PROGRAM BA02PL_LineBackground
VAR
END_VAR

MAIN.stLine_BA02PL.fbLine(stLine:=MAIN.stLine_BA02PL,bMainLine:=TRUE);
MAIN.stLine_BA02PL.stStation_BA02PL01.fbStation(
				stLine:=MAIN.stLine_BA02PL,
				stStation:=MAIN.stLine_BA02PL.stStation_BA02PL01);
MAIN.stLine_BA02PL.stStation_BA02PL02.fbStation(
				stLine:=MAIN.stLine_BA02PL,
				stStation:=MAIN.stLine_BA02PL.stStation_BA02PL02);
MAIN.stLine_BA02PL.stStation_BA02PL03.fbStation(
				stLine:=MAIN.stLine_BA02PL,
				stStation:=MAIN.stLine_BA02PL.stStation_BA02PL03);
MAIN.stLine_BA02PL.stStation_BA02PL04.fbStation(
				stLine:=MAIN.stLine_BA02PL,
				stStation:=MAIN.stLine_BA02PL.stStation_BA02PL04);
MAIN.stLine_BA02PL.stStation_BA02PL05.fbStation( 
				stLine:=MAIN.stLine_BA02PL,
				stStation:=MAIN.stLine_BA02PL.stStation_BA02PL05);
MAIN.stLine_BA02PL.stStation_BA02PL06.fbStation(
				stLine:=MAIN.stLine_BA02PL,
				stStation:=MAIN.stLine_BA02PL.stStation_BA02PL06);
MAIN.stLine_BA02PL.stStation_BA02PL07.fbStation(
				stLine:=MAIN.stLine_BA02PL,
				stStation:=MAIN.stLine_BA02PL.stStation_BA02PL07);

END_PROGRAM

(* stored: Version 1.1.0.1, ProductVersion 3.1.4024.15
   POU BA02PL_LineBackground: Id {3c14947d-ab13-4a56-9101-d2239dd3d8ae}, SpecialFunc None *)
